TYPE ST_Safety_ToSafetyPrg :
STRUCT
	b_ErrorReset						: BOOL;
	b_EmergencyStopSoftwareOK			: BOOL;
	b_SafetyRunStop						: BOOL := TRUE;
	contactors							: ST_Safety_ContactorEDM;
END_STRUCT
END_TYPE

(* stored: Version 1.1.0.1, ProductVersion 3.1.4026.18
   DUT ST_Safety_ToSafetyPrg: Id {c156d6d5-b116-41ed-a3f0-4db4909da4a9} *)
